# EPICS substitutions: app/Db/eventDriver.substitutions
file eventDriver.template
{
    pattern
    { IOC,    RATE, PERIOD,         EVENT }
    { $(IOC), FAST, $(FAST_PERIOD),   2 }
    { $(IOC), MED,  $(MED_PERIOD),    3 }
    { $(IOC), SLOW, $(SLOW_PERIOD),   4 }
}
